// TIA Portal V21 export
// export: Created 2026-07-07T08:27:32.6446113Z, ExportSetting WithReadOnly, DisplayName Totally Integrated Automation Portal, DisplayVersion V21, DisplayName SINAMICS Startdrive Advanced, DisplayVersion V21, DisplayName SINAMICS Startdrive G110M, G120, G120C, G120D, G120P, G115D, DisplayVersion V21, DisplayName SINAMICS Startdrive G130, G150, S120, S150, G200, G220, S200, S210, S220, Innomotics MVD, DisplayVersion V21, DisplayName STEP 7 Professional, DisplayVersion V21, DisplayName STEP 7 Safety, DisplayVersion V21, DisplayName Tech WebApplication, DisplayVersion V21, DisplayName WinCC Basic/Comfort/Advanced, DisplayVersion V21, DisplayName WinCC Professional, DisplayVersion V21, DisplayName WinCC Unified, DisplayVersion V21
FUNCTION "FC_ModeInterlock_LAD" : Void   // FC2, LAD
{ S7_Optimized_Access := 'TRUE' }
// stored: CodeModifiedDate 2026-07-07T08:27:04.0853797Z, CompileDate 2026-07-07T08:27:05.4592799Z, CreationDate 2026-07-07T08:27:04.0611103Z, DownloadDate 0001-01-01T00:00:00Z, InterfaceModifiedDate 2026-07-07T08:27:04.0611103Z, IsConsistent true, LibraryConformanceStatus 警告： 该对象包含对全局数据块的访问。, LoadMemoryLength 10131, ModifiedDate 2026-07-07T08:27:04.2019708Z, PLCSimAdvancedSupport true, ParameterModified 2026-07-07T08:27:04.0611103Z, SetENOAutomatically false, StructureModified 2026-07-07T08:27:04.0611103Z, WorkMemoryLength 158
BEGIN

REGION Network 1: Communication normal
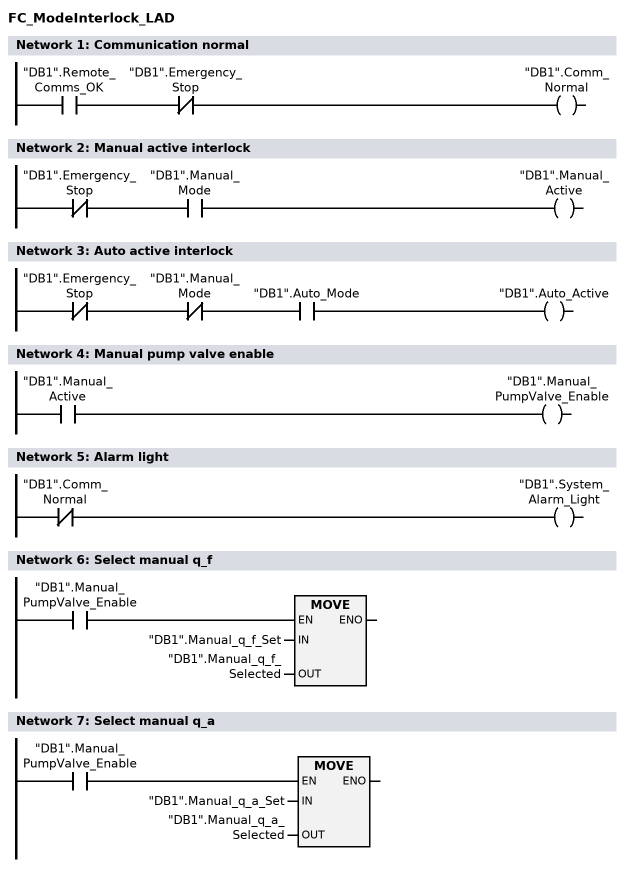
   RUNG wire#powerrail
      Contact( "DB1".Remote_Comms_OK )
      I_Contact( "DB1".Emergency_Stop )
      Coil( "DB1".Comm_Normal )
   END_RUNG
   // the same network as SCL:
   "DB1".Comm_Normal := "DB1".Remote_Comms_OK AND NOT "DB1".Emergency_Stop;
END_REGION

REGION Network 2: Manual active interlock
   RUNG wire#powerrail
      I_Contact( "DB1".Emergency_Stop )
      Contact( "DB1".Manual_Mode )
      Coil( "DB1".Manual_Active )
   END_RUNG
   // the same network as SCL:
   "DB1".Manual_Active := NOT "DB1".Emergency_Stop AND "DB1".Manual_Mode;
END_REGION

REGION Network 3: Auto active interlock
   RUNG wire#powerrail
      I_Contact( "DB1".Emergency_Stop )
      I_Contact( "DB1".Manual_Mode )
      Contact( "DB1".Auto_Mode )
      Coil( "DB1".Auto_Active )
   END_RUNG
   // the same network as SCL:
   "DB1".Auto_Active := NOT "DB1".Emergency_Stop AND NOT "DB1".Manual_Mode AND "DB1".Auto_Mode;
END_REGION

REGION Network 4: Manual pump valve enable
   RUNG wire#powerrail
      Contact( "DB1".Manual_Active )
      Coil( "DB1".Manual_PumpValve_Enable )
   END_RUNG
   // the same network as SCL:
   "DB1".Manual_PumpValve_Enable := "DB1".Manual_Active;
END_REGION

REGION Network 5: Alarm light
   RUNG wire#powerrail
      I_Contact( "DB1".Comm_Normal )
      Coil( "DB1".System_Alarm_Light )
   END_RUNG
   // the same network as SCL:
   "DB1".System_Alarm_Light := NOT "DB1".Comm_Normal;
END_REGION

REGION Network 6: Select manual q_f
   RUNG wire#powerrail
      Contact( "DB1".Manual_PumpValve_Enable )
      { S7_GenerateENO := "TRUE" } Move(in := "DB1".Manual_q_f_Set, out := "DB1".Manual_q_f_Selected)
   END_RUNG
   // the same network as SCL:
   IF "DB1".Manual_PumpValve_Enable THEN <??.?> := "DB1".Manual_q_f_Set; END_IF;
END_REGION

REGION Network 7: Select manual q_a
   RUNG wire#powerrail
      Contact( "DB1".Manual_PumpValve_Enable )
      { S7_GenerateENO := "TRUE" } Move(in := "DB1".Manual_q_a_Set, out := "DB1".Manual_q_a_Selected)
   END_RUNG
   // the same network as SCL:
   IF "DB1".Manual_PumpValve_Enable THEN <??.?> := "DB1".Manual_q_a_Set; END_IF;
END_REGION
END_FUNCTION
